FUNCTION_BLOCK LT_GT
VAR_INPUT
	INT_SOURCE_A: INT;
	INT_SOURCE_B: INT;
END_VAR
VAR_OUTPUT
	SIGNAL_BOOL: BOOL;
END_VAR
VAR
	M0: BOOL;
	M1: BOOL;
END_VAR

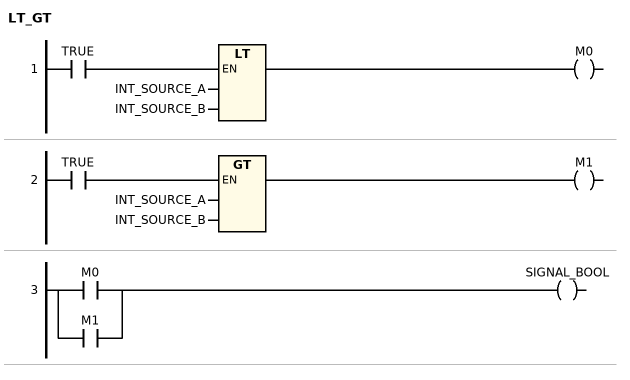
// NETWORK 1
M0 := INT_SOURCE_A < INT_SOURCE_B;

// NETWORK 2
M1 := INT_SOURCE_A > INT_SOURCE_B;

// NETWORK 3
SIGNAL_BOOL := M0 OR M1;

END_FUNCTION_BLOCK

(* stored: Version 1.1.0.1, ProductVersion 3.1.4024.12
   POU LT_GT: Id {af9f6031-0526-4e81-91ea-2ea1f2fd1618}, SpecialFunc None *)
